(* Logix 5000 project; controller R5_CSS vendor 1 type 14 code 74 rev 19.11; software revision 19.01; part 5 of 20 *)
(* tags used below, declared in another part *)
   AC102A : ANALYTICAL;   // QUENCH WATER CONDUCTIVITY CONTROL
   AlarmMaster : DINT;
   AlarmMasterDisable : BOOL;
   AlarmMasterResetTON : TIMER;
   AlarmResetPB : BOOL;
   ColdBoot : BOOL;
   DisableCommand : BOOL;
   EnableCommand : BOOL;
   Fault : BOOL;
   FC108 : FLOW_CONTROL;   // QUENCH FEED FLOW TRANSMITTER
   FC140A : FLOW_CONTROL;   // QUENCH TOWER UPPER SPRAY FLOW CONTROL
   FC140B : FLOW_CONTROL;   // QUENCH TOWER LOWER SPRAY FLOW CONTROL
   FireFlowAlarmFromUTL : BOOL;
   FirstScanLatch : BOOL;
   FirstScanLatchTON : TIMER;
   HART1 : HARTModuleDef;
   HARTData1 : HARTData;
   HMI_ShowReboot : BOOL;
   HMI_ShowRebootTmr : TIMER;
   Instrument_LOS : BOOL[32];
   IP_Address : DINT[4];
   IP_AddressGetMSG : MESSAGE;
   IP_AddressGetMSG_TON : TIMER;
   IP_AddressSetMSG : MESSAGE;
   LC205 : LEVEL_CONTROL;   // OVERHEAD CONDENSER BASIN LEVEL CONTROL
   LC302 : LEVEL_CONTROL;   // COALESCER OIL CHAMBER LEVEL CONTROL
   LC303A : LEVEL_CONTROL;   // AQUEOUS PHASE OF PRIMARY SETTLER
   My_IP_Address : DINT[4];
   My_Subnet : DINT[4];
   Option_F1_Occupancy : BOOL;   // STATUS FROM UTL PLC 0=DISABLED 1=ENABLED
   P101_OK_TON : TIMER;
   P101A : PUMP_CONTROL;
   P101A_OK : BOOL;
   P101B : PUMP_CONTROL;
   P101B_OK : BOOL;
   P302A : PUMP_CONTROL;
   P302B : PUMP_CONTROL;
   P303_OK_TON : TIMER;
   P303A : PUMP_CONTROL;
   P303A_OK : BOOL;
   P303B : PUMP_CONTROL;
   P303B_OK : BOOL;
   PC101A : PRESSURE_CONTROL;   // LOWER QUENCH TOWER PRESSURE TRANSMITTER
   PC101B : PRESSURE_CONTROL;   // UPPER QUENCH TOWER PRESSURE TRANSMITTER PRESSURE CONTOL
   PC407B : PRESSURE_CONTROL;   // POST HX LOW PRESSURE TRANSMITTER
   SetMyIP_Enabled : BOOL;
   TC101A : TEMP_CONTROL;   // QUENCH BASIN TRANSFER BASIN A TEMPERATURE CONTROL
   TC108 : TEMP_CONTROL;   // QUENCH TOWER EXIT GAS TEMPERATURE CONTROL
   TC114A : TEMP_CONTROL;   // QUENCH BASIN SHELL TEMPERATURE CONTROL
   TCP_GetAll : TCPGetAllConfig;
   TCP_SetAll : TCPSetAllConfig;
   UTL_Comms : DINT[3];
   UTL_CommsLossAlm : BOOL;
   WarmBoot : BOOL;
(* MainProgram, continued *)

ROUTINE A2c_HART_WRITEE   (* ladder *)
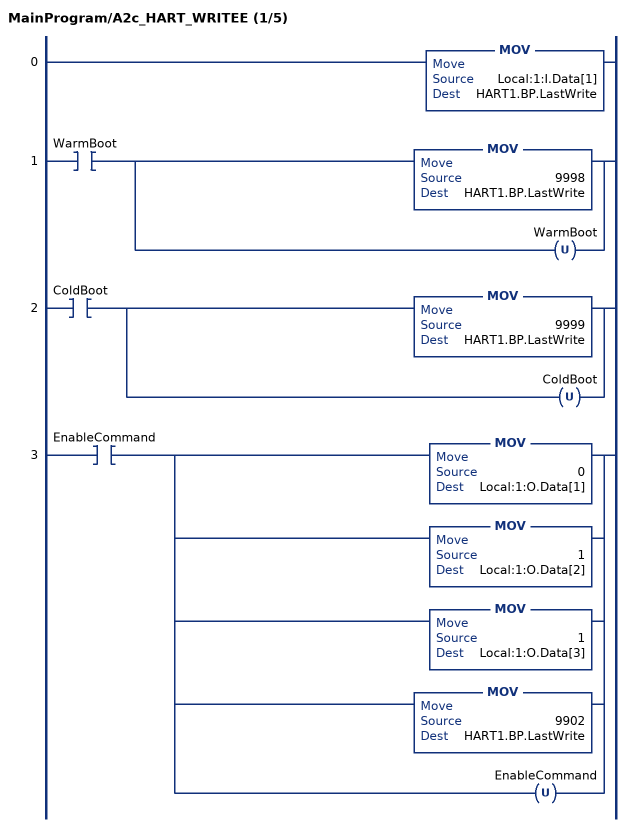
   0: MOV(Local:1:I.Data[1],HART1.BP.LastWrite);
   1: XIC(WarmBoot)[MOV(9998,HART1.BP.LastWrite) ,OTU(WarmBoot) ];
   2: XIC(ColdBoot)[MOV(9999,HART1.BP.LastWrite) ,OTU(ColdBoot) ];
   3: XIC(EnableCommand)[MOV(0,Local:1:O.Data[1]) ,MOV(1,Local:1:O.Data[2]) ,MOV(1,Local:1:O.Data[3]) ,MOV(9902,HART1.BP.LastWrite) ,OTU(EnableCommand) ];
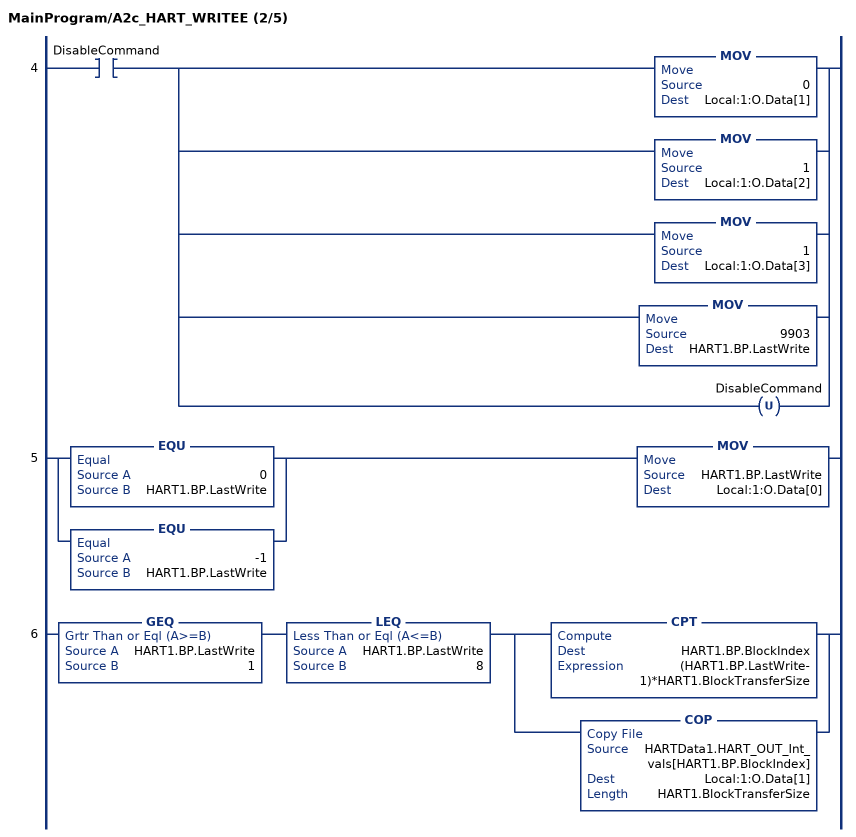
   4: XIC(DisableCommand)[MOV(0,Local:1:O.Data[1]) ,MOV(1,Local:1:O.Data[2]) ,MOV(1,Local:1:O.Data[3]) ,MOV(9903,HART1.BP.LastWrite) ,OTU(DisableCommand) ];
   5: [EQU(0,HART1.BP.LastWrite) ,EQU(-1,HART1.BP.LastWrite) ]MOV(HART1.BP.LastWrite,Local:1:O.Data[0]);
   6: GEQ(HART1.BP.LastWrite,1)LEQ(HART1.BP.LastWrite,8)[CPT(HART1.BP.BlockIndex,(HART1.BP.LastWrite-1)*HART1.BlockTransferSize) ,COP(HARTData1.HART_OUT_Int_vals[HART1.BP.BlockIndex],Local:1:O.Data[1],HART1.BlockTransferSize) ];
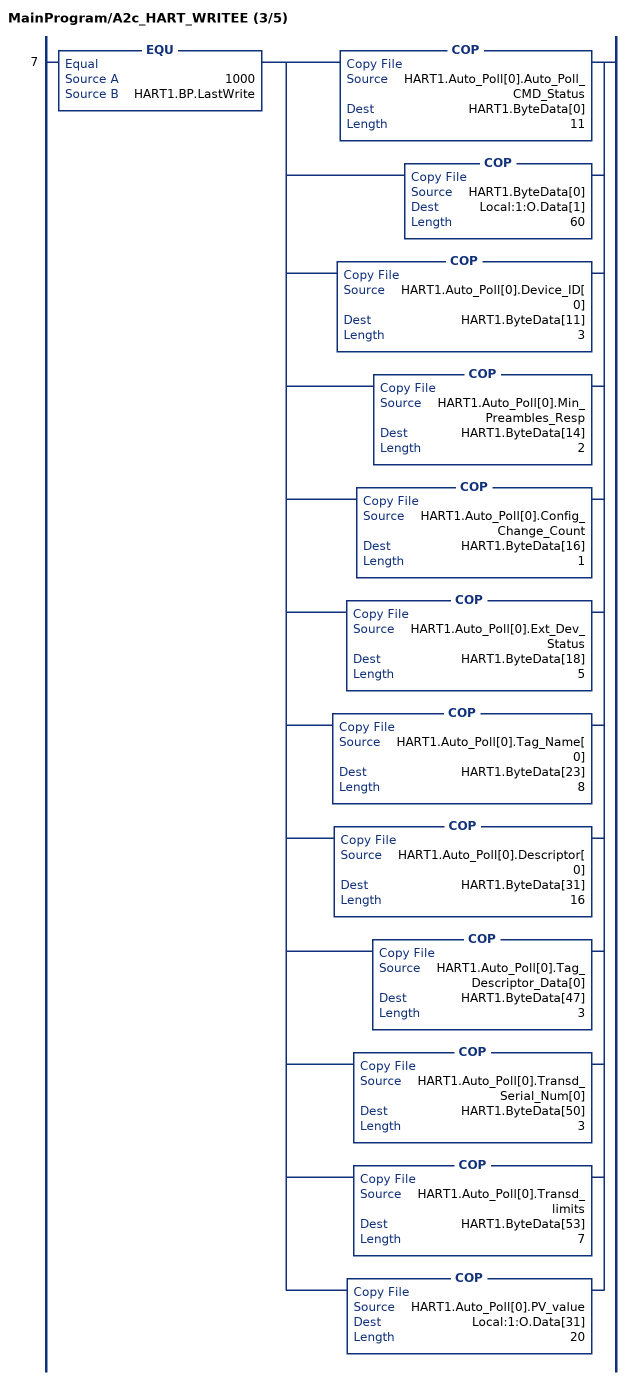
   7: EQU(1000,HART1.BP.LastWrite)[COP(HART1.Auto_Poll[0].Auto_Poll_CMD_Status,HART1.ByteData[0],11) ,COP(HART1.ByteData[0],Local:1:O.Data[1],60) ,COP(HART1.Auto_Poll[0].Device_ID[0],HART1.ByteData[11],3) ,COP(HART1.Auto_Poll[0].Min_Preambles_Resp,HART1.ByteData[14],2) ,COP(HART1.Auto_Poll[0].Config_Change_Count,HART1.ByteData[16],1) ,COP(HART1.Auto_Poll[0].Ext_Dev_Status,HART1.ByteData[18],5) ,COP(HART1.Auto_Poll[0].Tag_Name[0],HART1.ByteData[23],8) ,COP(HART1.Auto_Poll[0].Descriptor[0],HART1.ByteData[31],16) ,COP(HART1.Auto_Poll[0].Tag_Descriptor_Data[0],HART1.ByteData[47],3) ,COP(HART1.Auto_Poll[0].Transd_Serial_Num[0],HART1.ByteData[50],3) ,COP(HART1.Auto_Poll[0].Transd_limits,HART1.ByteData[53],7) ,COP(HART1.Auto_Poll[0].PV_value,Local:1:O.Data[31],20) ];
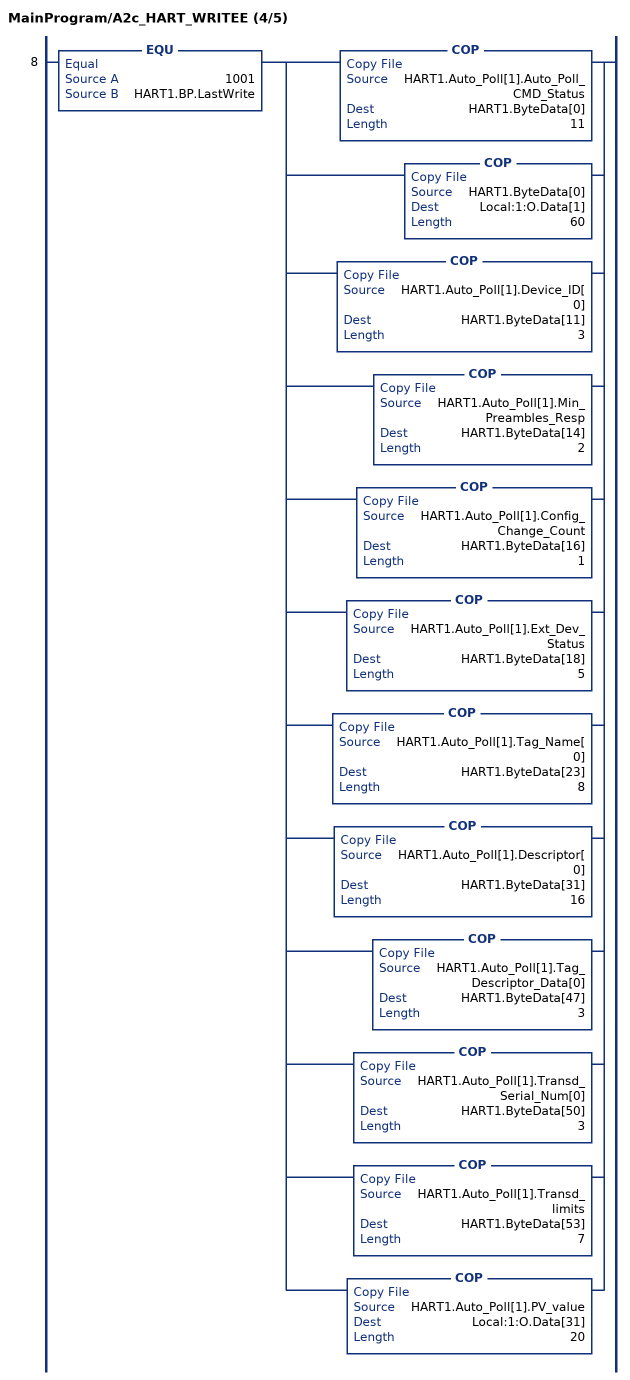
   8: EQU(1001,HART1.BP.LastWrite)[COP(HART1.Auto_Poll[1].Auto_Poll_CMD_Status,HART1.ByteData[0],11) ,COP(HART1.ByteData[0],Local:1:O.Data[1],60) ,COP(HART1.Auto_Poll[1].Device_ID[0],HART1.ByteData[11],3) ,COP(HART1.Auto_Poll[1].Min_Preambles_Resp,HART1.ByteData[14],2) ,COP(HART1.Auto_Poll[1].Config_Change_Count,HART1.ByteData[16],1) ,COP(HART1.Auto_Poll[1].Ext_Dev_Status,HART1.ByteData[18],5) ,COP(HART1.Auto_Poll[1].Tag_Name[0],HART1.ByteData[23],8) ,COP(HART1.Auto_Poll[1].Descriptor[0],HART1.ByteData[31],16) ,COP(HART1.Auto_Poll[1].Tag_Descriptor_Data[0],HART1.ByteData[47],3) ,COP(HART1.Auto_Poll[1].Transd_Serial_Num[0],HART1.ByteData[50],3) ,COP(HART1.Auto_Poll[1].Transd_limits,HART1.ByteData[53],7) ,COP(HART1.Auto_Poll[1].PV_value,Local:1:O.Data[31],20) ];
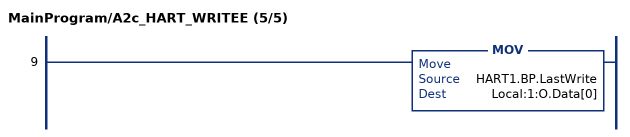
   9: MOV(HART1.BP.LastWrite,Local:1:O.Data[0]);
END_ROUTINE

ROUTINE A3_ENET_STATUS   (* ladder *)
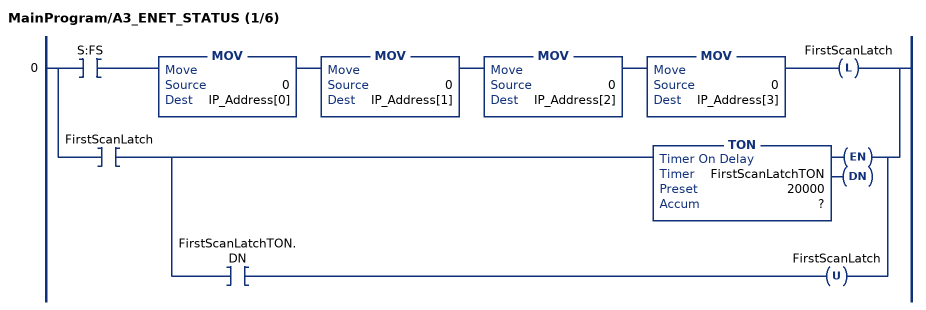
   0: [XIC(S:FS) MOV(0,IP_Address[0]) MOV(0,IP_Address[1]) MOV(0,IP_Address[2]) MOV(0,IP_Address[3]) OTL(FirstScanLatch) ,XIC(FirstScanLatch) [TON(FirstScanLatchTON,?,?) ,XIC(FirstScanLatchTON.DN) OTU(FirstScanLatch) ] ];
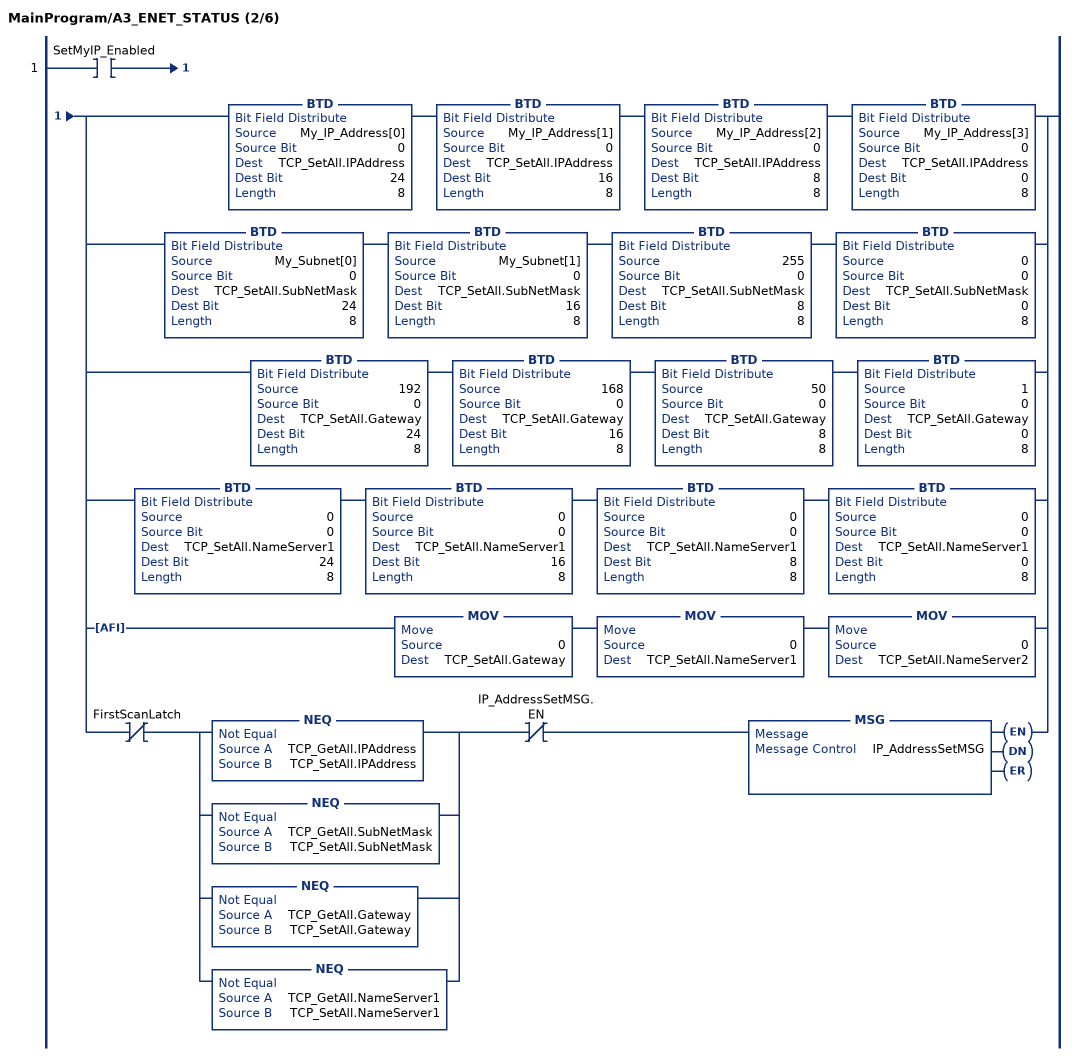
   1: XIC(SetMyIP_Enabled)[BTD(My_IP_Address[0],0,TCP_SetAll.IPAddress,24,8) BTD(My_IP_Address[1],0,TCP_SetAll.IPAddress,16,8) BTD(My_IP_Address[2],0,TCP_SetAll.IPAddress,8,8) BTD(My_IP_Address[3],0,TCP_SetAll.IPAddress,0,8) ,BTD(My_Subnet[0],0,TCP_SetAll.SubNetMask,24,8) BTD(My_Subnet[1],0,TCP_SetAll.SubNetMask,16,8) BTD(255,0,TCP_SetAll.SubNetMask,8,8) BTD(0,0,TCP_SetAll.SubNetMask,0,8) ,BTD(192,0,TCP_SetAll.Gateway,24,8) BTD(168,0,TCP_SetAll.Gateway,16,8) BTD(50,0,TCP_SetAll.Gateway,8,8) BTD(1,0,TCP_SetAll.Gateway,0,8) ,BTD(0,0,TCP_SetAll.NameServer1,24,8) BTD(0,0,TCP_SetAll.NameServer1,16,8) BTD(0,0,TCP_SetAll.NameServer1,8,8) BTD(0,0,TCP_SetAll.NameServer1,0,8) ,AFI() MOV(0,TCP_SetAll.Gateway) MOV(0,TCP_SetAll.NameServer1) MOV(0,TCP_SetAll.NameServer2) ,XIO(FirstScanLatch) [NEQ(TCP_GetAll.IPAddress,TCP_SetAll.IPAddress) ,NEQ(TCP_GetAll.SubNetMask,TCP_SetAll.SubNetMask) ,NEQ(TCP_GetAll.Gateway,TCP_SetAll.Gateway) ,NEQ(TCP_GetAll.NameServer1,TCP_SetAll.NameServer1) ] XIO(IP_AddressSetMSG.EN) MSG(IP_AddressSetMSG) ];
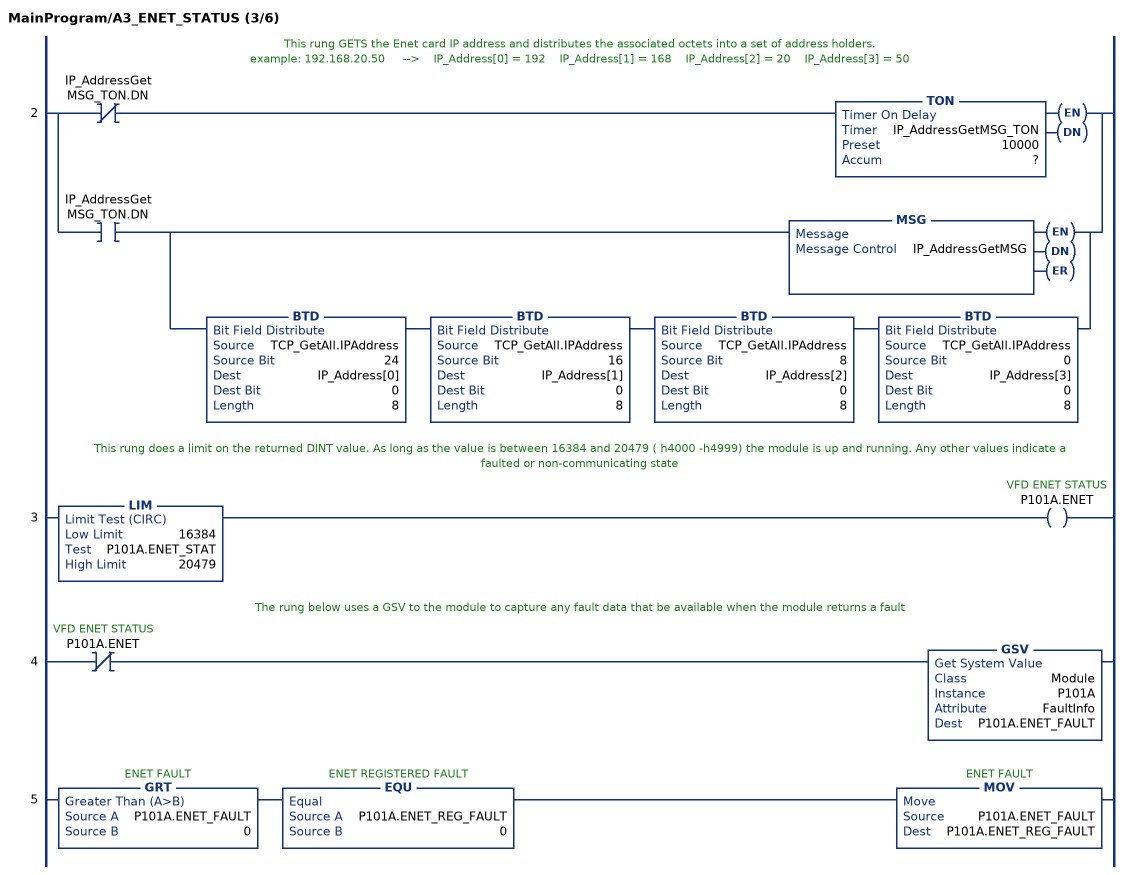
   // This rung GETS the Enet card IP address and distributes the associated octets into a set of address holders.
   // example: 192.168.20.50     -->    IP_Address[0] = 192    IP_Address[1] = 168    IP_Address[2] = 20    IP_Address[3] = 50
   2: [XIO(IP_AddressGetMSG_TON.DN) TON(IP_AddressGetMSG_TON,?,?) ,XIC(IP_AddressGetMSG_TON.DN) [MSG(IP_AddressGetMSG) ,BTD(TCP_GetAll.IPAddress,24,IP_Address[0],0,8) BTD(TCP_GetAll.IPAddress,16,IP_Address[1],0,8) BTD(TCP_GetAll.IPAddress,8,IP_Address[2],0,8) BTD(TCP_GetAll.IPAddress,0,IP_Address[3],0,8) ] ];
   // This rung does a limit on the returned DINT value. As long as the value is between 16384 and 20479 ( h4000 -h4999) the module is up and running. Any other values indicate a faulted or non-communicating state
   3: LIM(16384,P101A.ENET_STAT,20479)OTE(P101A.ENET);
   // The rung below uses a GSV to the module to capture any fault data that be available when the module returns a fault
   4: XIO(P101A.ENET)GSV(Module,P101A,FaultInfo,P101A.ENET_FAULT);
   5: GRT(P101A.ENET_FAULT,0)EQU(P101A.ENET_REG_FAULT,0)MOV(P101A.ENET_FAULT,P101A.ENET_REG_FAULT);
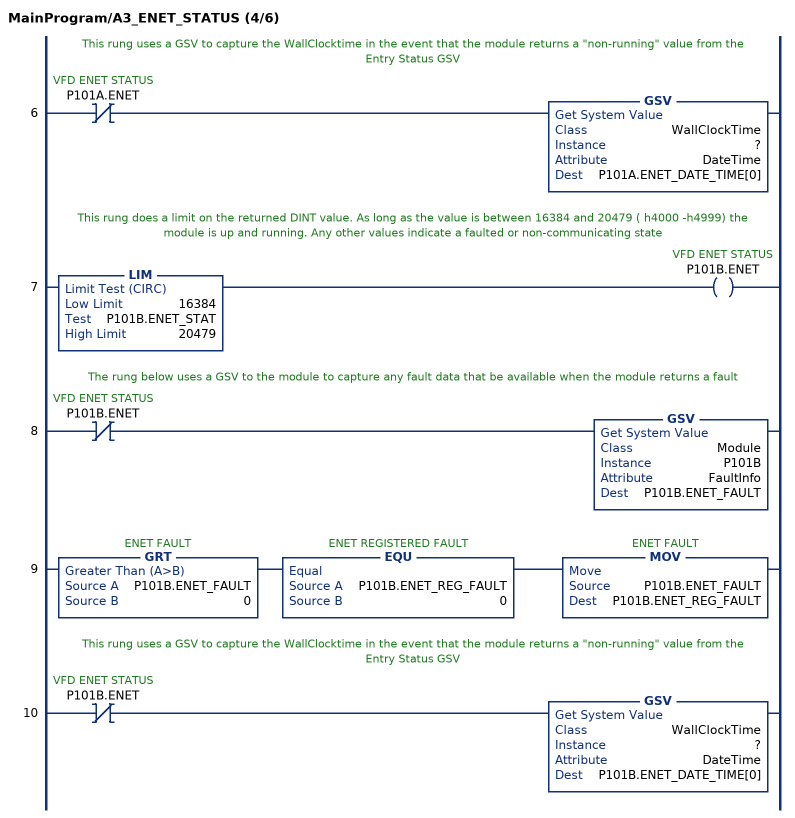
   // This rung uses a GSV to capture the WallClocktime in the event that the module returns a "non-running" value from the Entry Status GSV
   6: XIO(P101A.ENET)GSV(WallClockTime,?,DateTime,P101A.ENET_DATE_TIME[0]);
   // This rung does a limit on the returned DINT value. As long as the value is between 16384 and 20479 ( h4000 -h4999) the module is up and running. Any other values indicate a faulted or non-communicating state
   7: LIM(16384,P101B.ENET_STAT,20479)OTE(P101B.ENET);
   // The rung below uses a GSV to the module to capture any fault data that be available when the module returns a fault
   8: XIO(P101B.ENET)GSV(Module,P101B,FaultInfo,P101B.ENET_FAULT);
   9: GRT(P101B.ENET_FAULT,0)EQU(P101B.ENET_REG_FAULT,0)MOV(P101B.ENET_FAULT,P101B.ENET_REG_FAULT);
   // This rung uses a GSV to capture the WallClocktime in the event that the module returns a "non-running" value from the Entry Status GSV
   10: XIO(P101B.ENET)GSV(WallClockTime,?,DateTime,P101B.ENET_DATE_TIME[0]);
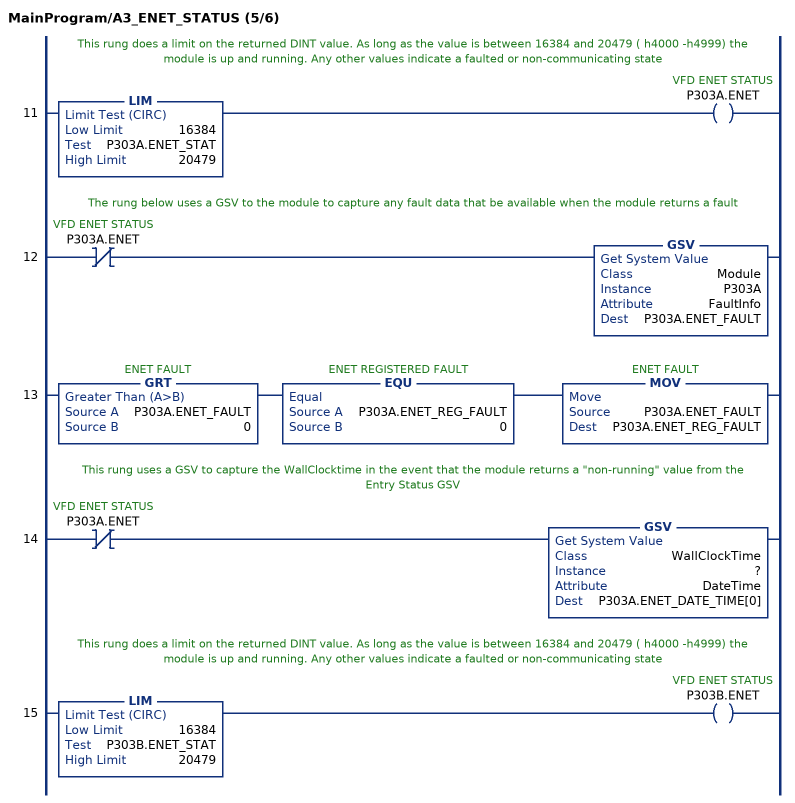
   // This rung does a limit on the returned DINT value. As long as the value is between 16384 and 20479 ( h4000 -h4999) the module is up and running. Any other values indicate a faulted or non-communicating state
   11: LIM(16384,P303A.ENET_STAT,20479)OTE(P303A.ENET);
   // The rung below uses a GSV to the module to capture any fault data that be available when the module returns a fault
   12: XIO(P303A.ENET)GSV(Module,P303A,FaultInfo,P303A.ENET_FAULT);
   13: GRT(P303A.ENET_FAULT,0)EQU(P303A.ENET_REG_FAULT,0)MOV(P303A.ENET_FAULT,P303A.ENET_REG_FAULT);
   // This rung uses a GSV to capture the WallClocktime in the event that the module returns a "non-running" value from the Entry Status GSV
   14: XIO(P303A.ENET)GSV(WallClockTime,?,DateTime,P303A.ENET_DATE_TIME[0]);
   // This rung does a limit on the returned DINT value. As long as the value is between 16384 and 20479 ( h4000 -h4999) the module is up and running. Any other values indicate a faulted or non-communicating state
   15: LIM(16384,P303B.ENET_STAT,20479)OTE(P303B.ENET);
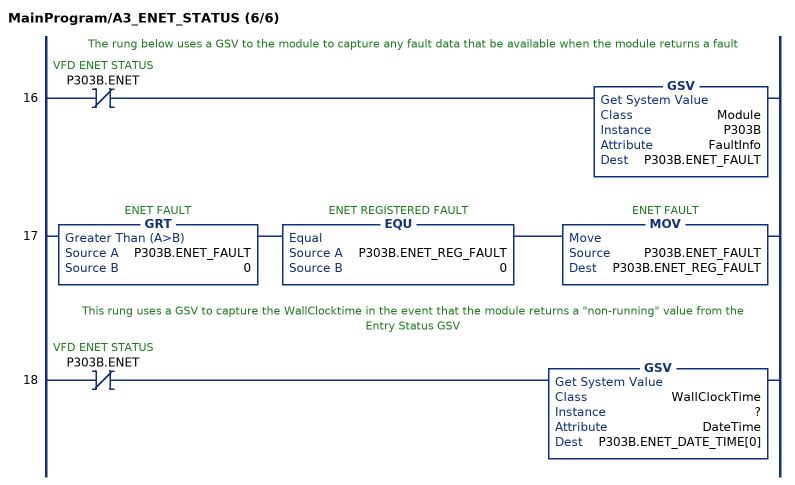
   // The rung below uses a GSV to the module to capture any fault data that be available when the module returns a fault
   16: XIO(P303B.ENET)GSV(Module,P303B,FaultInfo,P303B.ENET_FAULT);
   17: GRT(P303B.ENET_FAULT,0)EQU(P303B.ENET_REG_FAULT,0)MOV(P303B.ENET_FAULT,P303B.ENET_REG_FAULT);
   // This rung uses a GSV to capture the WallClocktime in the event that the module returns a "non-running" value from the Entry Status GSV
   18: XIO(P303B.ENET)GSV(WallClockTime,?,DateTime,P303B.ENET_DATE_TIME[0]);
END_ROUTINE

ROUTINE A4_Alarms_General   (* ladder *)
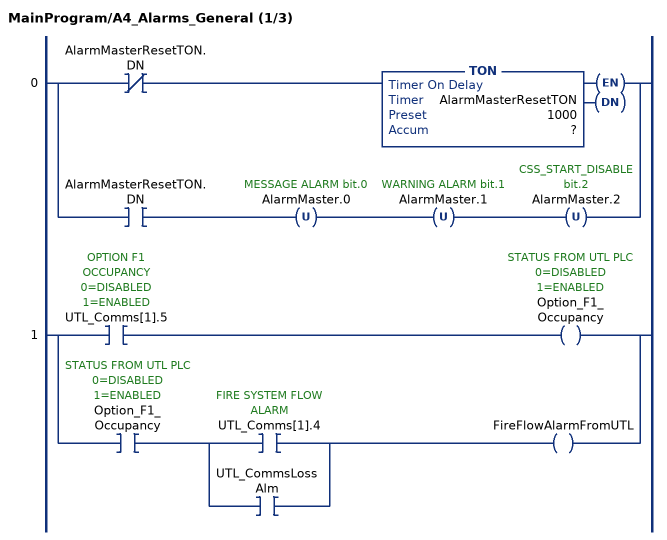
   0: [XIO(AlarmMasterResetTON.DN) TON(AlarmMasterResetTON,?,?) ,XIC(AlarmMasterResetTON.DN) OTU(AlarmMaster.0) OTU(AlarmMaster.1) OTU(AlarmMaster.2) ];
   1: [XIC(UTL_Comms[1].5) OTE(Option_F1_Occupancy) ,XIC(Option_F1_Occupancy) [XIC(UTL_Comms[1].4) ,XIC(UTL_CommsLossAlm) ] OTE(FireFlowAlarmFromUTL) ];
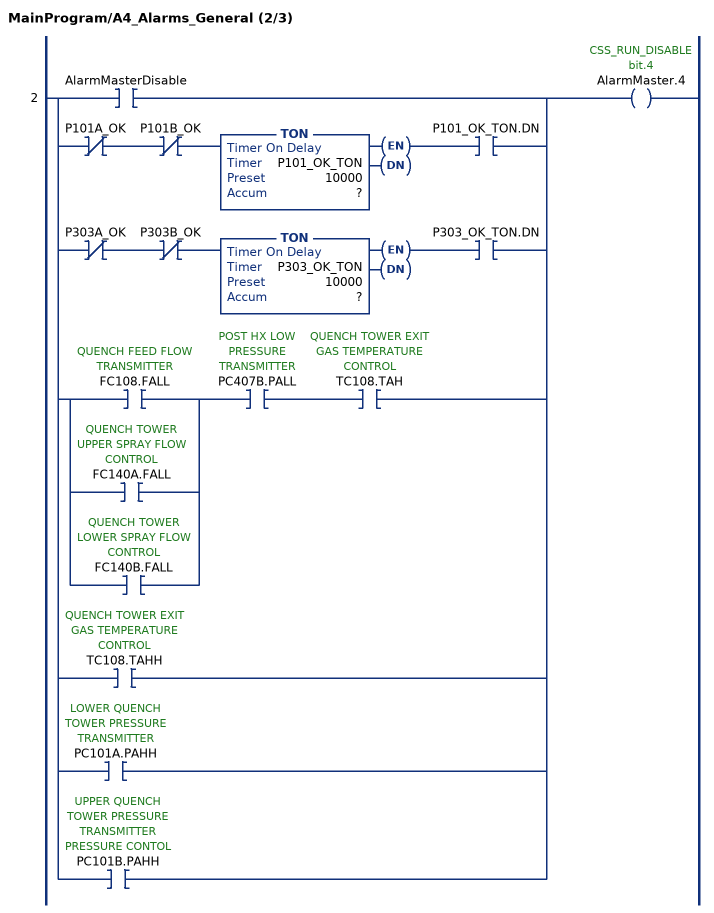
   2: [XIC(AlarmMasterDisable) ,XIO(P101A_OK) XIO(P101B_OK) TON(P101_OK_TON,?,?) XIC(P101_OK_TON.DN) ,XIO(P303A_OK) XIO(P303B_OK) TON(P303_OK_TON,?,?) XIC(P303_OK_TON.DN) ,[XIC(FC108.FALL) ,XIC(FC140A.FALL) ,XIC(FC140B.FALL) ] XIC(PC407B.PALL) XIC(TC108.TAH) ,XIC(TC108.TAHH) ,XIC(PC101A.PAHH) ,XIC(PC101B.PAHH) ]OTE(AlarmMaster.4);
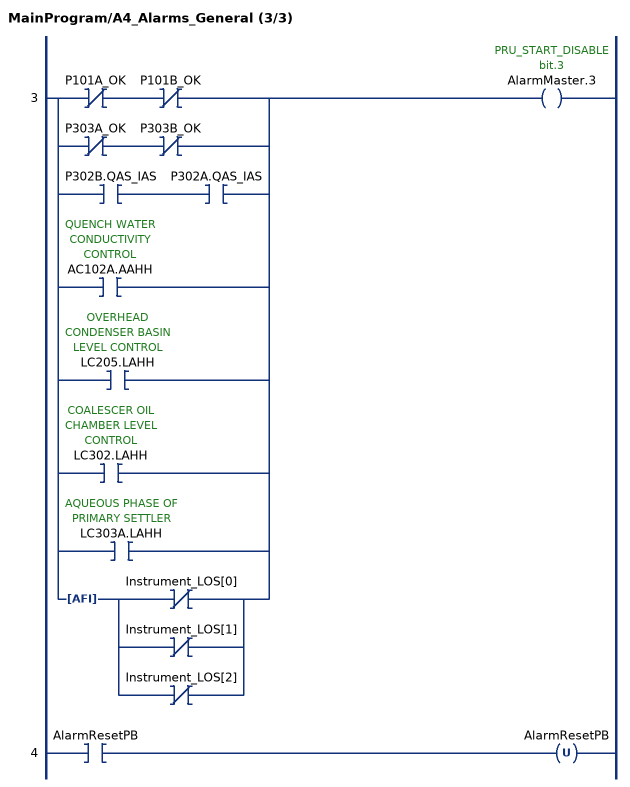
   3: [XIO(P101A_OK) XIO(P101B_OK) ,XIO(P303A_OK) XIO(P303B_OK) ,XIC(P302B.QAS_IAS) XIC(P302A.QAS_IAS) ,XIC(AC102A.AAHH) ,XIC(LC205.LAHH) ,XIC(LC302.LAHH) ,XIC(LC303A.LAHH) ,AFI() [XIO(Instrument_LOS[0]) ,XIO(Instrument_LOS[1]) ,XIO(Instrument_LOS[2]) ] ]OTE(AlarmMaster.3);
   4: XIC(AlarmResetPB)OTU(AlarmResetPB);
END_ROUTINE

ROUTINE A5a_LOAD_START_UP_PARAMETERS   (* ladder *)
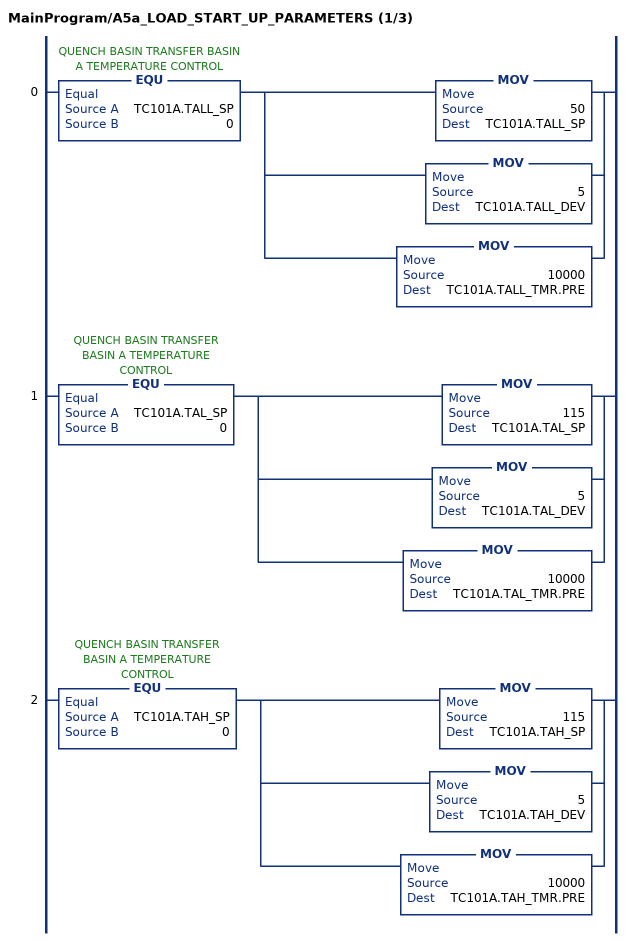
   0: EQU(TC101A.TALL_SP,0)[MOV(50,TC101A.TALL_SP) ,MOV(5,TC101A.TALL_DEV) ,MOV(10000,TC101A.TALL_TMR.PRE) ];
   1: EQU(TC101A.TAL_SP,0)[MOV(115,TC101A.TAL_SP) ,MOV(5,TC101A.TAL_DEV) ,MOV(10000,TC101A.TAL_TMR.PRE) ];
   2: EQU(TC101A.TAH_SP,0)[MOV(115,TC101A.TAH_SP) ,MOV(5,TC101A.TAH_DEV) ,MOV(10000,TC101A.TAH_TMR.PRE) ];
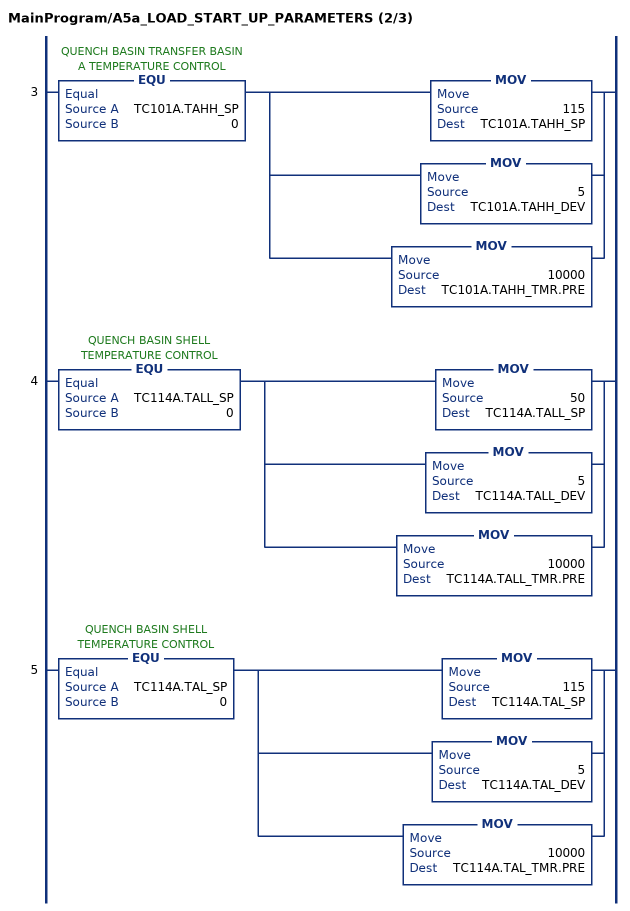
   3: EQU(TC101A.TAHH_SP,0)[MOV(115,TC101A.TAHH_SP) ,MOV(5,TC101A.TAHH_DEV) ,MOV(10000,TC101A.TAHH_TMR.PRE) ];
   4: EQU(TC114A.TALL_SP,0)[MOV(50,TC114A.TALL_SP) ,MOV(5,TC114A.TALL_DEV) ,MOV(10000,TC114A.TALL_TMR.PRE) ];
   5: EQU(TC114A.TAL_SP,0)[MOV(115,TC114A.TAL_SP) ,MOV(5,TC114A.TAL_DEV) ,MOV(10000,TC114A.TAL_TMR.PRE) ];
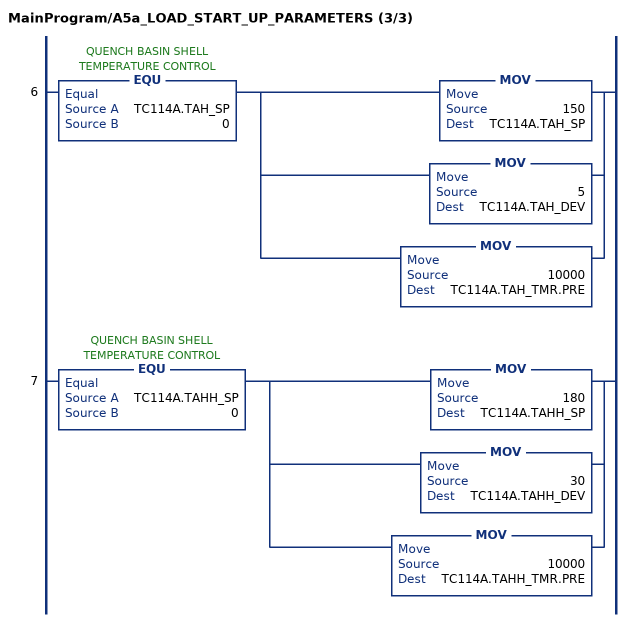
   6: EQU(TC114A.TAH_SP,0)[MOV(150,TC114A.TAH_SP) ,MOV(5,TC114A.TAH_DEV) ,MOV(10000,TC114A.TAH_TMR.PRE) ];
   7: EQU(TC114A.TAHH_SP,0)[MOV(180,TC114A.TAHH_SP) ,MOV(30,TC114A.TAHH_DEV) ,MOV(10000,TC114A.TAHH_TMR.PRE) ];
END_ROUTINE

ROUTINE A5b_LOCAL_HMI   (* ladder *)
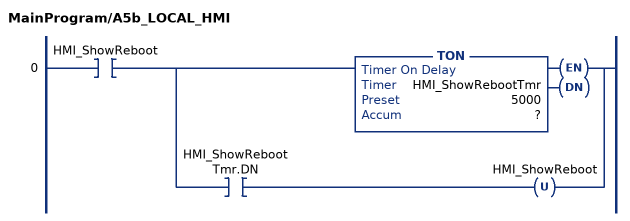
   0: XIC(HMI_ShowReboot)[TON(HMI_ShowRebootTmr,?,?) ,XIC(HMI_ShowRebootTmr.DN) OTU(HMI_ShowReboot) ];
END_ROUTINE
